// Common base class for the "Get" requests
TYPE ST_AlpacaGetRequest :
STRUCT
    sName       : STRING;
    eStatusCode : E_AlpacaStatusCode;
    rAge        : REAL;                 // age of the last reading, in seconds, since the last loop start
END_STRUCT
END_TYPE

(* stored: Version 1.1.0.1, ProductVersion 3.1.4024.12
   DUT ST_AlpacaGetRequest: Id {f724c27b-bc6b-400b-8f79-e57d55e14056} *)
